Fanuc KAREL source: IO0035.KL

PROGRAM IO0035
%NOLOCKGROUP
ROUTINE RTEST
VAR
L1 : ARRAY[3] OF INTEGER;L2 : XYZWPR
L3 : JOINTPOS9
L4 : POSITION
A:INTEGER
B:REAL
C:REAL
D:BOOLEAN
E:REAL
BEGIN
--
A=1
L1[1]=2
D=TRUE
E=1.0
DOUT[L1[A]]=TRUE
END RTEST
BEGIN
RTEST
END IO0035
